// Monitors the baseplate chiller from the flow sensor
FUNCTION_BLOCK FB_BaseplateChiller
VAR_INPUT
	bBaseplateChillerFlow : BOOL; // Signal from the flow sensor. Normally high.
END_VAR
VAR_OUTPUT
	{attribute 'pytmc' := '
		pv: ERROR
		io: i
		field: OSV MAJOR
		field: ZSV NO_ALARM
		field: ZNAM OK
		field: ONAM ERROR
	'}
	bError : BOOL; // Whether an error was detected. Should latch until reset
END_VAR
VAR
END_VAR

IF NOT bBaseplateChillerFlow THEN
	bError := TRUE;
END_IF

// Reset latched errors
METHOD Reset
VAR_INPUT
END_VAR
bError := FALSE;
END_METHOD

END_FUNCTION_BLOCK

(* stored: Version 1.1.0.1, ProductVersion 3.1.4020.14
   POU FB_BaseplateChiller: Id {b3f0a1a0-251e-4592-bbae-0313baecaf1e}, SpecialFunc None
   Method Reset: Id {93053126-6c32-4761-a872-242edc24bfe8} *)
